// POUs/FB_NVRAM_Manager
FUNCTION_BLOCK FB_NVRAM_Manager
VAR_INPUT
    VI_Command                  : BYTE; // 1=WRITE, 2=READ, 3=FORMAT
    VI_RecordIndex              : INT;
    VI_DataPtr                  : POINTER TO BYTE;
    VI_DataSize                 : UDINT; // КРИТИЧНО: используем этот размер вместо SIZEOF
    VI_System_Time_MS           : UDINT;
    VI_Operator_ID              : STRING(10);
    VI_IsActivePLC              : BOOL;
    VI_TwoPersonConfirmation    : BOOL;
END_VAR
VAR_OUTPUT
    VO_Done                     : BOOL;
    VO_Error                    : UDINT;
    VO_ErrorID                  : UDINT;
    VO_ReadDataPtr              : POINTER TO BYTE;
    VO_HMI_Status_Message       : STRING(200);
END_VAR
VAR
    L_state                     : BYTE;
    L_step                      : UDINT;
    L_temp_buffer               : ARRAY[1..132] OF BYTE;
    L_crc32                     : FB_CRC32_Calculator;
    L_confirm_start_time        : UDINT;
    L_cmd_copy                  : BYTE;
    L_prev_Command              : BYTE;
    L_i                         : UDINT;
    L_current_time              : UDINT;
    L_cmd_rising                : BOOL;
    L_data_crc                  : DWORD;
    L_FileHandle                : RTS_IEC_HANDLE;
    L_FileName                  : STRING := '/home/root/nvram_data.bin';
    L_FileResult                : RTS_IEC_RESULT;
    L_BytesProcessed            : UDINT;
    L_BackupIdx                 : INT := 1; // Для ротации
    L_Offset                    : DINT;
END_VAR
VAR CONSTANT
    C_MAGIC_NUMBER              : UDINT := 16#534D5254; // "SMRT"
    C_STRUCT_VERSION            : UINT := 21; // ТЗ v21.0
    C_NVRAM_BASE_ADDR           : UDINT := 16#20000;
    C_HEADER_SIZE               : UDINT := 12;
    C_RECORD_SIZE               : UDINT := 128;
    C_RECORD_TOTAL_SIZE         : UDINT := 132;
    C_MAX_RECORDS               : UDINT := 96;
    C_TWO_PERSON_TIMEOUT_MS     : UDINT := 120000;
END_VAR

// Логика выполнения
L_current_time := VI_System_Time_MS;

// Детекция фронта команды
L_cmd_rising := (VI_Command <> 0) AND (L_prev_Command = 0);
L_prev_Command := VI_Command;

CASE L_state OF
    0: // ОЖИДАНИЕ (IDLE)
        IF L_cmd_rising THEN
            VO_Done := FALSE;
            VO_Error := 0;
            
            // Валидация индекса
            IF (VI_RecordIndex < 1) OR (TO_UDINT(VI_RecordIndex) > C_MAX_RECORDS) THEN
                VO_Error := 16#1501;
                VO_HMI_Status_Message := 'NVRAM: Неверный индекс записи';
                VO_Done := TRUE;
                RETURN;
            END_IF;

            // Валидация указателя
            IF VI_DataPtr = 0 THEN
                VO_Error := 16#150A;
                VO_HMI_Status_Message := 'NVRAM: Нулевой указатель данных';
                VO_Done := TRUE;
                RETURN;
            END_IF;

            IF VI_Command = 1 THEN // ЗАПИСЬ (WRITE)
                IF NOT VI_IsActivePLC THEN
                    VO_Error := 16#1509;
                    VO_HMI_Status_Message := 'NVRAM: Запись запрещена (STANDBY)';
                    VO_Done := TRUE;
                ELSIF VI_DataSize > C_RECORD_SIZE THEN
                    VO_Error := 16#150B;
                    VO_HMI_Status_Message := 'NVRAM: Размер данных больше 128 байт';
                    VO_Done := TRUE;
                ELSE
                    L_state := 1; // Переход к записи
                    L_step := 0;
                END_IF;
            ELSIF VI_Command = 2 THEN // ЧТЕНИЕ (READ)
                L_state := 2; // Переход к чтению
                L_step := 0;
            END_IF;
        END_IF;

    1: // ЗАПИСЬ_ЗАПИСИ (WRITE_RECORD)
        CASE L_step OF
            0: // Подготовка буфера и расчет CRC
                FOR L_i := 0 TO C_RECORD_SIZE - 1 DO
                    IF L_i < VI_DataSize THEN
                        L_temp_buffer[TO_INT(L_i + 1)] := VI_DataPtr[TO_INT(L_i)];
                    ELSE
                        L_temp_buffer[TO_INT(L_i + 1)] := 16#00;
                    END_IF;
                END_FOR;
                L_data_crc := L_crc32.Calculate(ADR(L_temp_buffer[1]), C_RECORD_SIZE);
                L_step := 1;
                
            1: // Открытие файла для записи
                L_FileHandle := SysFileOpen(L_FileName, AM_WRITE, ADR(L_FileResult));
                IF L_FileResult = 0 THEN
                    L_step := 2;
                ELSE
                    VO_Error := 16#150C;
                    L_state := 0;
                END_IF;
                
            2: // Позиционирование и запись
                L_Offset := TO_DINT(VI_RecordIndex - 1) * TO_DINT(C_RECORD_TOTAL_SIZE);
                L_FileResult := SysFileSetPos(L_FileHandle, TO_UDINT(L_Offset));
                L_BytesProcessed := TO_UDINT(SysFileWrite(L_FileHandle, ADR(L_temp_buffer[1]), TO_UDINT(C_RECORD_TOTAL_SIZE), ADR(L_FileResult)));
                L_FileResult := SysFileClose(L_FileHandle);
                VO_Done := TRUE;
                L_state := 0;
        END_CASE;

    2: // ЧТЕНИЕ_ЗАПИСИ (READ_RECORD)
        CASE L_step OF
            0: // Открытие файла для чтения
                L_FileHandle := SysFileOpen(L_FileName, AM_READ, ADR(L_FileResult));
                IF L_FileResult = 0 THEN
                    L_step := 1;
                ELSE
                    VO_Error := 16#150D;
                    L_state := 0;
                END_IF;
                
            1: // Чтение данных
                L_Offset := TO_DINT(VI_RecordIndex - 1) * TO_DINT(C_RECORD_TOTAL_SIZE);
                L_FileResult := SysFileSetPos(L_FileHandle, TO_UDINT(L_Offset));
                L_BytesProcessed := TO_UDINT(SysFileRead(L_FileHandle, ADR(L_temp_buffer[1]), TO_UDINT(C_RECORD_TOTAL_SIZE), ADR(L_FileResult)));
                L_FileResult := SysFileClose(L_FileHandle);
                
                // Копирование в выходной указатель
                FOR L_i := 0 TO C_RECORD_SIZE - 1 DO
                    IF L_i < VI_DataSize THEN
                        VI_DataPtr[TO_INT(L_i)] := L_temp_buffer[TO_INT(L_i + 1)];
                    END_IF;
                END_FOR;
                VO_ReadDataPtr := VI_DataPtr;
                VO_Done := TRUE;
                L_state := 0;
        END_CASE;
END_CASE;

END_FUNCTION_BLOCK

// POUs/FB_CRC32_Calculator
FUNCTION_BLOCK FB_CRC32_Calculator
VAR
    L_Table : ARRAY[0..255] OF DWORD;
    L_Initialized : BOOL := FALSE;
    L_i : INT;
    L_j : INT;
    L_Entry : DWORD;
END_VAR

METHOD Calculate : DWORD
VAR_INPUT
    VI_DataPtr : POINTER TO BYTE;
    VI_Size : UDINT;
END_VAR
VAR
    L_k : UDINT;
    L_CRC : DWORD := 16#FFFFFFFF;
END_VAR
InitTable();

IF VI_DataPtr = 0 OR VI_Size = 0 THEN
    Calculate := 0;
    RETURN;
END_IF;

FOR L_k := 0 TO VI_Size - 1 DO
    L_CRC := L_Table[TO_INT((L_CRC XOR VI_DataPtr[TO_INT(L_k)]) AND 16#FF)] XOR SHR(L_CRC, 8);
END_FOR;

Calculate := L_CRC XOR 16#FFFFFFFF;
END_METHOD

METHOD PRIVATE InitTable
VAR_INPUT
END_VAR
IF L_Initialized THEN RETURN; END_IF;

FOR L_i := 0 TO 255 DO
    L_Entry := TO_DWORD(L_i);
    FOR L_j := 0 TO 7 DO
        IF (L_Entry AND 1) <> 0 THEN
            L_Entry := SHR(L_Entry, 1) XOR 16#EDB88320;
        ELSE
            L_Entry := SHR(L_Entry, 1);
        END_IF;
    END_FOR;
    L_Table[L_i] := L_Entry;
END_FOR;
L_Initialized := TRUE;
END_METHOD

END_FUNCTION_BLOCK

// POUs/FB_Gateway_Interface
FUNCTION_BLOCK FB_Gateway_Interface
VAR_INPUT
    VI_System_Time_MS           : UDINT;
    VI_Local_PLC_Role           : E_PLC_ROLE;
    VI_Incoming_Command         : ST_Gateway_Command;
    VI_Command_Received         : BOOL;
    
    // Состояния системы
    VI_FloorHeating_Temps       : ARRAY[1..16] OF REAL;
    VI_Room_Temps               : ARRAY[1..16] OF REAL;
    VI_Zone_Valve_States        : ARRAY[1..16] OF BOOL;
    VI_Manifold_Pressures       : ARRAY[1..5] OF REAL;
    VI_Manifold_Pump_States     : ARRAY[1..5] OF BOOL;
    VI_Outdoor_Temp             : REAL;
    VI_Security_Armed           : BOOL;
    VI_Flood_Alarm_Active       : BOOL;
    VI_Gas_Alarm_Active         : BOOL;
    VI_Fire_Alarm_Active        : BOOL;
    VI_Methane_Concentration    : REAL;
    VI_Lighting_Base_Levels     : ARRAY[1..16] OF BYTE;
    VI_Socket_States            : ARRAY[1..36] OF BOOL;
    VI_Blinds_Positions         : ARRAY[1..20] OF BYTE;
    VI_Active_Scenario          : E_SCENARIO_TYPE;
END_VAR

VAR_OUTPUT
    VO_Modbus_Registers         : ARRAY[0..200] OF WORD; // Расширенный диапазон
    VO_Lighting_Override        : ARRAY[1..16] OF BYTE;
    VO_Socket_Override          : ARRAY[1..36] OF BOOL;
    VO_Data_Ready               : BOOL;
    VO_HMI_Status_Message       : STRING(200);
END_VAR

VAR
    L_last_update_time          : UDINT;
    L_i                         : INT;
    L_j                         : INT;
    L_idx                       : INT;
    L_tmp_word                  : WORD;
END_VAR

// Обновление данных Modbus (раз в 1 сек)
IF (VI_System_Time_MS - L_last_update_time) >= 1000 THEN
    L_last_update_time := VI_System_Time_MS;
    
    // 0: Статус ПЛК и Аварии
    L_tmp_word := 0;
    IF VI_Local_PLC_Role = E_PLC_ROLE.ROLE_ACTIVE THEN L_tmp_word := L_tmp_word OR 1; END_IF;
    IF VI_Security_Armed THEN L_tmp_word := L_tmp_word OR 2; END_IF;
    IF VI_Flood_Alarm_Active THEN L_tmp_word := L_tmp_word OR 4; END_IF;
    IF VI_Gas_Alarm_Active THEN L_tmp_word := L_tmp_word OR 8; END_IF;
    IF VI_Fire_Alarm_Active THEN L_tmp_word := L_tmp_word OR 16; END_IF;
    VO_Modbus_Registers[0] := L_tmp_word;

    // 1-16: Температуры пола (x10)
    FOR L_i := 1 TO 16 DO
        VO_Modbus_Registers[L_i] := TO_WORD(TO_INT(VI_FloorHeating_Temps[L_i] * 10.0));
    END_FOR;

    // 17-32: Температуры помещений (x10)
    FOR L_i := 1 TO 16 DO
        VO_Modbus_Registers[16 + L_i] := TO_WORD(TO_INT(VI_Room_Temps[L_i] * 10.0));
    END_FOR;

    // 33: Состояние клапанов зон (битовая маска 1-16)
    L_tmp_word := 0;
    FOR L_i := 1 TO 16 DO
        IF VI_Zone_Valve_States[L_i] THEN
            L_tmp_word := L_tmp_word OR SHL(TO_WORD(1), L_i - 1);
        END_IF;
    END_FOR;
    VO_Modbus_Registers[33] := L_tmp_word;

    // 34-38: Давление в коллекторах (x100)
    FOR L_i := 1 TO 5 DO
        VO_Modbus_Registers[33 + L_i] := TO_WORD(TO_INT(VI_Manifold_Pressures[L_i] * 100.0));
    END_FOR;

    // 40-55: Базовое освещение
    FOR L_i := 1 TO 16 DO
        VO_Modbus_Registers[39 + L_i] := TO_WORD(VI_Lighting_Base_Levels[L_i]);
    END_FOR;

    // 60-79: Положение штор (20 шт)
    FOR L_i := 1 TO 20 DO
        VO_Modbus_Registers[59 + L_i] := TO_WORD(VI_Blinds_Positions[L_i]);
    END_FOR;

    // 80-82: Розетки (битовая маска, 36 розеток -> 3 WORD)
    FOR L_i := 0 TO 2 DO
        L_tmp_word := 0;
        FOR L_j := 1 TO 16 DO
            L_idx := (L_i * 16) + L_j;
            IF L_idx <= 36 THEN
                IF VI_Socket_States[L_idx] THEN
                    L_tmp_word := L_tmp_word OR SHL(TO_WORD(1), L_j - 1);
                END_IF;
            END_IF;
        END_FOR;
        VO_Modbus_Registers[79 + L_i] := L_tmp_word;
    END_FOR;

    VO_Data_Ready := TRUE;
END_IF;

// Обработка входящих команд
IF VI_Command_Received AND (VI_Local_PLC_Role = E_PLC_ROLE.ROLE_ACTIVE) THEN
    CASE VI_Incoming_Command.command_type OF
        1: // Управление сценариями
            GVL_Vars.G_Current_Scenario := VI_Incoming_Command.target_scenario;
            VO_HMI_Status_Message := 'Gateway: Сценарий изменен';
        2: // Управление освещением
            IF (VI_Incoming_Command.target_zone >= 1) AND (VI_Incoming_Command.target_zone <= 16) THEN
                VO_Lighting_Override[VI_Incoming_Command.target_zone] := TO_BYTE(VI_Incoming_Command.target_value);
                VO_HMI_Status_Message := 'Gateway: Команда освещения принята';
            END_IF;
        3: // Розетки
            IF (VI_Incoming_Command.target_zone >= 1) AND (VI_Incoming_Command.target_zone <= 36) THEN
                VO_Socket_Override[VI_Incoming_Command.target_zone] := VI_Incoming_Command.target_on_off;
            END_IF;
        4: // Охрана
            // Логика постановки/снятия через PIN в FB_Security_System_Manager
            // Здесь можно только передать запрос
            VO_HMI_Status_Message := 'Gateway: Запрос охраны принят';
    END_CASE;
END_IF;

END_FUNCTION_BLOCK

// POUs/FB_Debug_Logger
FUNCTION_BLOCK FB_Debug_Logger
VAR_INPUT
    VI_Config           : ST_Debug_Logger_Config;
    VI_System_Time_MS   : UDINT;
    VI_Floor_Temps      : ARRAY[1..16] OF REAL;
    VI_Pump_Currents    : ARRAY[1..5] OF REAL;
    VI_Error_Code       : UDINT;
END_VAR
VAR
    L_buffer            : ARRAY[1..1000] OF ST_Debug_Log_Record;
    L_write_idx         : INT := 1;
    L_last_log_time     : UDINT;
    L_i                 : INT;
END_VAR

// Цикл логирования
IF VI_Config.enabled AND (VI_System_Time_MS - L_last_log_time >= VI_Config.sampling_period_ms) THEN
    L_last_log_time := VI_System_Time_MS;
    
    // Логируем температуры (если изменились или по таймауту)
    FOR L_i := 1 TO 16 DO
        L_buffer[L_write_idx].timestamp_ms := VI_System_Time_MS;
        L_buffer[L_write_idx].level := E_Debug_Log_Level.LOG_LEVEL_VERBOSE;
        L_buffer[L_write_idx].source_id := TO_BYTE(L_i);
        L_buffer[L_write_idx].value_real := VI_Floor_Temps[L_i];
        L_buffer[L_write_idx].text := 'Floor Temp Update';
        
        L_write_idx := (L_write_idx MOD 1000) + 1;
    END_FOR;

    // Логируем ошибки
    IF VI_Error_Code <> 0 THEN
        L_buffer[L_write_idx].timestamp_ms := VI_System_Time_MS;
        L_buffer[L_write_idx].level := E_Debug_Log_Level.LOG_LEVEL_MINIMAL;
        L_buffer[L_write_idx].event_code := TO_WORD(VI_Error_Code);
        L_buffer[L_write_idx].text := 'System Error Detected';
        L_write_idx := (L_write_idx MOD 1000) + 1;
    END_IF;
END_IF;

END_FUNCTION_BLOCK

// PLC_A/Application/PRG_PLC_B
PROGRAM PRG_PLC_B
VAR
    L_PLC_ID : BYTE := 2;
END_VAR

// Для ПЛК B: если он активен, G_Active_PLC_ID := 2
PRG_Main();

END_PROGRAM

// IValveController
INTERFACE IValveController

METHOD CloseValve : BOOL
VAR_INPUT
    VI_Operator_ID : STRING(10);
    VI_Force : BOOL;
END_VAR
END_METHOD

METHOD GetStatus : BYTE
VAR_INPUT
END_VAR
END_METHOD

METHOD OpenValve : BOOL
VAR_INPUT
    VI_Operator_ID : STRING(10);
    VI_Force : BOOL;
END_VAR
END_METHOD

END_INTERFACE

// POUs/FB_AccessCode_Manager
FUNCTION_BLOCK FB_AccessCode_Manager
VAR_INPUT
    VI_System_Time_MS : UDINT;
    VI_IsActivePLC    : BOOL;
    VI_Code_To_Check  : STRING(4);
END_VAR
VAR_OUTPUT
    VO_Code_Valid     : BOOL;
END_VAR
VAR
    L_Codes : ARRAY[1..5] OF STRING(4) := ['1234', '5678', '0000', '1111', '2222'];
    L_i : INT;
END_VAR

VO_Code_Valid := FALSE;
FOR L_i := 1 TO 5 DO
    IF L_Codes[L_i] = VI_Code_To_Check THEN
        VO_Code_Valid := TRUE;
        RETURN;
    END_IF;
END_FOR;

END_FUNCTION_BLOCK

// POUs/FB_Astro_Timer
FUNCTION_BLOCK FB_Astro_Timer
VAR_INPUT
    VI_System_Time_MS : UDINT;
    VI_Latitude : REAL := 55.75; // Москва
    VI_Longitude : REAL := 37.61;
END_VAR
VAR_OUTPUT
    VO_Sunset_Time : TOD;
    VO_Sunrise_Time : TOD;
    VO_Is_Night : BOOL;
END_VAR
VAR
    L_Current_TOD : TOD;
END_VAR

// Упрощенная логика астро-таймера (ТЗ 15.2)
// В реальном проекте используется библиотека SysTimeRtc или расчет по формулам
L_Current_TOD := UDINT_TO_TOD(VI_System_Time_MS MOD 86400000);

// Примерные значения для средней полосы
VO_Sunrise_Time := TOD#06:00;
VO_Sunset_Time := TOD#18:00;

// ТЗ 15.2: Закат + 30 мин / Рассвет - 30 мин
VO_Is_Night := (L_Current_TOD > (VO_Sunset_Time + T#30m)) OR (L_Current_TOD < (VO_Sunrise_Time - T#30m));

END_FUNCTION_BLOCK

// POUs/FB_BlackBox_Recorder
FUNCTION_BLOCK FB_BlackBox_Recorder
VAR_INPUT
    VI_Current_Data : ST_BlackBox_Record;
    VI_Freeze       : BOOL;
END_VAR
VAR
    L_Write_Index   : INT := 0;
    L_FileHandle    : RTS_IEC_HANDLE;
    L_FileName      : STRING := '/home/root/blackbox_dump.bin';
    L_FileResult    : RTS_IEC_RESULT;
    L_State         : INT;
END_VAR

CASE L_State OF
    0: // Циклическая запись
        IF NOT G_BlackBox_Frozen THEN
            G_BlackBox_Buffer[L_Write_Index] := VI_Current_Data;
            G_BlackBox_LastIndex := L_Write_Index;
            
            L_Write_Index := L_Write_Index + 1;
            IF L_Write_Index > 99 THEN
                L_Write_Index := 0;
            END_IF;
            
            IF VI_Freeze THEN
                G_BlackBox_Frozen := TRUE;
                L_State := 1;
            END_IF;
        END_IF;
        
    1: // Сохранение на Flash (SD-карту или внутреннюю память ПЛК210)
        L_FileHandle := SysFileOpen(L_FileName, AM_WRITE, ADR(L_FileResult));
        IF L_FileResult = 0 THEN
            SysFileWrite(L_FileHandle, ADR(G_BlackBox_Buffer[0]), SIZEOF(G_BlackBox_Buffer), ADR(L_FileResult));
            SysFileClose(L_FileHandle);
            L_State := 2;
        END_IF;
        
    2: // Завершено
        ;
END_CASE;

END_FUNCTION_BLOCK

// POUs/FB_Boiler_Cascade_Controller
FUNCTION_BLOCK FB_Boiler_Cascade_Controller
VAR_INPUT
    VI_Demand_kW : REAL;
    VI_IsActivePLC : BOOL;
END_VAR
VAR_OUTPUT
    VO_Boiler1_On : BOOL;
    VO_Boiler2_On : BOOL;
END_VAR
VAR
    L_Lead_Boiler : BYTE := 1; // 1 или 2
    L_Boiler1_Hours : UDINT;
    L_Boiler2_Hours : UDINT;
    L_Last_Hour_Update : UDINT;
    L_System_Time : UDINT;
END_VAR
VAR_INPUT
    VI_System_Time : UDINT;
END_VAR

// Логика ротации по наработке
IF (VI_System_Time - L_Last_Hour_Update) >= 3600000 THEN // Раз в час
    L_Last_Hour_Update := VI_System_Time;
    IF VO_Boiler1_On THEN L_Boiler1_Hours := L_Boiler1_Hours + 1; END_IF;
    IF VO_Boiler2_On THEN L_Boiler2_Hours := L_Boiler2_Hours + 1; END_IF;
    
    // Смена ведущего, если разница более 100 часов
    IF (L_Boiler1_Hours > L_Boiler2_Hours + 100) THEN
        L_Lead_Boiler := 2;
    ELSIF (L_Boiler2_Hours > L_Boiler1_Hours + 100) THEN
        L_Lead_Boiler := 1;
    END_IF;
END_IF;

IF VI_IsActivePLC THEN
    IF VI_Demand_kW > 24.0 THEN
        VO_Boiler1_On := TRUE;
        VO_Boiler2_On := TRUE;
    ELSIF VI_Demand_kW > 2.0 THEN
        VO_Boiler1_On := (L_Lead_Boiler = 1);
        VO_Boiler2_On := (L_Lead_Boiler = 2);
    ELSE
        VO_Boiler1_On := FALSE;
        VO_Boiler2_On := FALSE;
    END_IF;
END_IF;

END_FUNCTION_BLOCK

// POUs/FB_Boiler_Cascade_Manager
FUNCTION_BLOCK FB_Boiler_Cascade_Manager
VAR_INPUT
    VI_Boiler1_Status : ST_Boiler_Status;
    VI_Boiler2_Status : ST_Boiler_Status;
    VI_Role_Swap_Interval : UDINT := 168; // часы
END_VAR
VAR_OUTPUT
    VO_Boiler1_Enable : BOOL;
    VO_Boiler2_Enable : BOOL;
END_VAR

// Логика п. 2.8: Включение резервного при >80% мощности или отказе
IF VI_Boiler1_Status.Error OR VI_Boiler1_Status.Current_Power > 80.0 THEN
    VO_Boiler2_Enable := TRUE;
ELSE
    VO_Boiler2_Enable := FALSE;
END_IF;

VO_Boiler1_Enable := NOT VI_Boiler1_Status.Error;

END_FUNCTION_BLOCK

// POUs/FB_Calibration_Manager
FUNCTION_BLOCK FB_Calibration_Manager
VAR_INPUT
    VI_Raw_Value : REAL;
    VI_Type : BYTE; // 1-Temp, 2-Pressure, 3-Gas
    VI_Calib_Record : ST_Sensor_Calibration_Record;
    VI_System_Time_MS : UDINT;
    VI_Start_Verification : BOOL;
END_VAR
VAR_OUTPUT
    VO_Calibrated_Value : REAL;
    VO_Verification_Active : BOOL;
    VO_Verification_Failed : BOOL;
    VO_Deviation_Percent : REAL;
END_VAR
VAR
    L_Verification_Timer : TON;
    L_Initial_Value : REAL;
END_VAR

// 1. Расчет калиброванного значения
CASE VI_Type OF
    1: VO_Calibrated_Value := VI_Raw_Value + VI_Calib_Record.offset;
    2, 3: VO_Calibrated_Value := (VI_Raw_Value * VI_Calib_Record.multiplier) + VI_Calib_Record.offset;
END_CASE;

// 2. Верификация через 1 час (ТЗ 9.5)
IF VI_Start_Verification AND NOT VO_Verification_Active THEN
    VO_Verification_Active := TRUE;
    L_Initial_Value := VO_Calibrated_Value;
    L_Verification_Timer(IN := TRUE, PT := T#1h);
END_IF;

L_Verification_Timer(IN := VO_Verification_Active);

IF L_Verification_Timer.Q THEN
    VO_Verification_Active := FALSE;
    L_Verification_Timer(IN := FALSE);
    
    // ТЗ 9.5: Отклонение ≤2.0% (норма) / >5.0% (ошибка)
    IF L_Initial_Value <> 0 THEN
        VO_Deviation_Percent := ABS(VO_Calibrated_Value - L_Initial_Value) / L_Initial_Value * 100.0;
    ELSE
        VO_Deviation_Percent := 0.0;
    END_IF;
    
    VO_Verification_Failed := (VO_Deviation_Percent > 5.0);
END_IF;

END_FUNCTION_BLOCK

// POUs/FB_CO_Detector
FUNCTION_BLOCK FB_CO_Detector
VAR_INPUT
    VI_CO_PPM : REAL;
    VI_Threshold_Warning : REAL := 30.0;
    VI_Threshold_Alarm   : REAL := 70.0;
END_VAR
VAR_OUTPUT
    VO_Warning_Active : BOOL;
    VO_Alarm_Active   : BOOL;
END_VAR

VO_Warning_Active := (VI_CO_PPM >= VI_Threshold_Warning);
VO_Alarm_Active := (VI_CO_PPM >= VI_Threshold_Alarm);

END_FUNCTION_BLOCK

// POUs/FB_Device_Predictive_Diag
FUNCTION_BLOCK FB_Device_Predictive_Diag
VAR_INPUT
    VI_Current_Value : REAL;      // Текущий ток или время
    VI_Nominal_Value : REAL;      // Эталонное значение
    VI_Is_Running    : BOOL;
    VI_Reset_Stats   : BOOL;
END_VAR
VAR_IN_OUT
    VIO_Health_Data  : ST_Device_Health;
END_VAR
VAR
    L_Prev_Running   : BOOL;
    L_Current_Sum    : REAL;
    L_Sample_Count   : UDINT;
END_VAR

// 1. Счётчик пусков и замер пускового тока
IF VI_Is_Running AND NOT L_Prev_Running THEN
    VIO_Health_Data.Starts_Count := VIO_Health_Data.Starts_Count + 1;
    VIO_Health_Data.Last_Start_Current := VI_Current_Value;
    
    // Обновление среднего пускового тока
    L_Sample_Count := L_Sample_Count + 1;
    L_Current_Sum := L_Current_Sum + VI_Current_Value;
    VIO_Health_Data.Avg_Start_Current := L_Current_Sum / UDINT_TO_REAL(L_Sample_Count);
END_IF;

// 2. Анализ отклонения (п. 12.1 ТЗ)
IF VI_Is_Running THEN
    // Если ток выше номинала на 50% - снижаем здоровье
    IF VI_Current_Value > (VI_Nominal_Value * 1.5) THEN
        IF VIO_Health_Data.Health_Score > 0 THEN
            VIO_Health_Data.Health_Score := VIO_Health_Data.Health_Score - 1;
        END_IF;
    END_IF;
END_IF;

// 3. Генерация предупреждения
IF VIO_Health_Data.Health_Score < 20 THEN
    VIO_Health_Data.Maintenance_Required := TRUE;
    VIO_Health_Data.Warning_Message := 'Критический износ: проверьте механику';
ELSIF VIO_Health_Data.Health_Score < 60 THEN
    VIO_Health_Data.Warning_Message := 'Предупреждение: повышенное трение';
END_IF;

L_Prev_Running := VI_Is_Running;

END_FUNCTION_BLOCK

// POUs/FB_Emergency_Valve_Open
FUNCTION_BLOCK FB_Emergency_Valve_Open
VAR_INPUT
    VI_Fire_Alarm : BOOL;
    VI_Gas_Alarm  : BOOL;
END_VAR
VAR_OUTPUT
    VO_Open_Cmd   : BOOL;
END_VAR

// Приоритетное открытие при любой серьезной аварии
VO_Open_Cmd := VI_Fire_Alarm OR VI_Gas_Alarm;

END_FUNCTION_BLOCK

// POUs/FB_Exhaust_Ventilation_Controller
FUNCTION_BLOCK FB_Exhaust_Ventilation_Controller
VAR_INPUT
    VI_Humidity : REAL;
    VI_CO2      : REAL;
    VI_Config   : ST_Ventilation_Unit_Config;
END_VAR
VAR_OUTPUT
    VO_Fan_Speed : BYTE;
END_VAR

IF VI_Humidity > VI_Config.Threshold_Hum THEN
    VO_Fan_Speed := 100;
ELSIF VI_CO2 > 800.0 THEN
    VO_Fan_Speed := 70;
ELSE
    VO_Fan_Speed := 40;
END_IF;

END_FUNCTION_BLOCK

// POUs/FB_Flood_Detector
FUNCTION_BLOCK FB_Flood_Detector
VAR_INPUT
    VI_Sensors : ARRAY[1..12] OF BOOL;
    VI_IsActivePLC : BOOL;
END_VAR
VAR_OUTPUT
    VO_Flood_Alarm : BOOL;
    VO_Close_Valve_35 : BOOL;
    VO_Close_Valve_36 : BOOL;
END_VAR
VAR
    L_i : INT;
END_VAR

VO_Flood_Alarm := FALSE;
VO_Close_Valve_35 := FALSE;
VO_Close_Valve_36 := FALSE;

FOR L_i := 1 TO 12 DO
    IF VI_Sensors[L_i] THEN
        VO_Flood_Alarm := TRUE;
        IF VI_IsActivePLC THEN
            // Логика п. 4.2: Зона 2 (4-5) и Зона 3 (6-7) делят клапан 36
            IF L_i >= 4 AND L_i <= 7 THEN
                VO_Close_Valve_36 := TRUE;
            ELSIF L_i >= 1 AND L_i <= 3 THEN
                VO_Close_Valve_35 := TRUE;
            END_IF;
        END_IF;
    END_IF;
END_FOR;

END_FUNCTION_BLOCK

// POUs/FB_FloorHeating_Controller
FUNCTION_BLOCK FB_FloorHeating_Controller
VAR_INPUT
    VI_Current_Temp : REAL;
    VI_Config : ST_FloorHeating_Circuit_Config;
    VI_Tariff : ST_Tariff_Config;
    VI_Current_Hour : UINT;
    VI_IsActivePLC : BOOL;
END_VAR
VAR_OUTPUT
    VO_Pump_Run : BOOL;
    VO_Valve_Pos : REAL; // 0..10V
    VO_Effective_Setpoint : REAL;
END_VAR
VAR
    L_Is_Night : BOOL;
END_VAR

// 1. Определение активного тарифа
IF VI_Tariff.Enabled THEN
    IF VI_Tariff.Night_Start_Hour > VI_Tariff.Night_End_Hour THEN
        // Переход через полночь (например, 23:00 - 07:00)
        L_Is_Night := (VI_Current_Hour >= VI_Tariff.Night_Start_Hour) OR (VI_Current_Hour < VI_Tariff.Night_End_Hour);
    ELSE
        // В пределах одного дня
        L_Is_Night := (VI_Current_Hour >= VI_Tariff.Night_Start_Hour) AND (VI_Current_Hour < VI_Tariff.Night_End_Hour);
    END_IF;
ELSE
    L_Is_Night := FALSE;
END_IF;

// 2. Расчет эффективной уставки
VO_Effective_Setpoint := VI_Config.design_temp;
IF L_Is_Night THEN
    VO_Effective_Setpoint := VO_Effective_Setpoint + VI_Tariff.Boost_Delta;
END_IF;

// 3. Простая логика управления (гистерезис)
IF VI_IsActivePLC THEN
    IF VI_Current_Temp < (VO_Effective_Setpoint - 0.5) THEN
        VO_Pump_Run := TRUE;
        VO_Valve_Pos := 10.0;
    ELSIF VI_Current_Temp > (VO_Effective_Setpoint + 0.5) THEN
        VO_Pump_Run := FALSE;
        VO_Valve_Pos := 0.0;
    END_IF;
END_IF;

END_FUNCTION_BLOCK

// POUs/FB_FloorHeating_Freeze_Protection
FUNCTION_BLOCK FB_FloorHeating_Freeze_Protection
VAR_INPUT
    VI_Floor_Temps : ARRAY[1..16] OF REAL;
    VI_Outdoor_Temp : REAL;
    VI_Threshold : REAL := 7.0;
END_VAR
VAR_OUTPUT
    VO_Freeze_Alert : BOOL;
    VO_Pump_Force_On : BOOL;
END_VAR
VAR
    L_i : INT;
END_VAR

VO_Freeze_Alert := FALSE;
VO_Pump_Force_On := FALSE;

FOR L_i := 1 TO 16 DO
    IF VI_Floor_Temps[L_i] < VI_Threshold THEN
        VO_Freeze_Alert := TRUE;
        VO_Pump_Force_On := TRUE;
        RETURN;
    END_IF;
END_FOR;

IF VI_Outdoor_Temp < -5.0 THEN
    VO_Pump_Force_On := TRUE;
END_IF;

END_FUNCTION_BLOCK

// POUs/FB_FloorHeating_Overheat_Protection
FUNCTION_BLOCK FB_FloorHeating_Overheat_Protection
VAR_INPUT
    VI_Temps : ARRAY[1..16] OF REAL;
    VI_Threshold : REAL := 45.0;
END_VAR
VAR_OUTPUT
    VO_Overheat_Detected : BOOL;
    VO_Locked_Circuits : ARRAY[1..16] OF BOOL;
END_VAR
VAR
    L_i : INT;
END_VAR

VO_Overheat_Detected := FALSE;
FOR L_i := 1 TO 16 DO
    IF VI_Temps[L_i] > VI_Threshold THEN
        VO_Overheat_Detected := TRUE;
        VO_Locked_Circuits[L_i] := TRUE;
    END_IF;
END_FOR;

END_FUNCTION_BLOCK

// POUs/FB_Gas_Methane_Detector
FUNCTION_BLOCK FB_Gas_Methane_Detector
VAR_INPUT
    VI_Methane_LEL : REAL;
    VI_Threshold_Alarm : REAL := 20.0;
END_VAR
VAR_OUTPUT
    VO_Alarm_Active : BOOL;
    VO_Close_Valve  : BOOL;
END_VAR

VO_Alarm_Active := (VI_Methane_LEL >= VI_Threshold_Alarm);
VO_Close_Valve := VO_Alarm_Active;

END_FUNCTION_BLOCK

// POUs/FB_Gas_Valve_Controller
FUNCTION_BLOCK FB_Gas_Valve_Controller IMPLEMENTS IValveController
VAR_INPUT
    VI_System_Time : UDINT;
    VI_IsActivePLC : BOOL;
    VI_Gas_Alarm   : BOOL;
    VI_Config      : ST_Gas_Valve_Configuration;
END_VAR
VAR_OUTPUT
    VO_Valve_Closed : BOOL;
    VO_Status_Msg   : STRING(200);
END_VAR

// При аварии газа - немедленное закрытие
IF VI_Gas_Alarm AND VI_IsActivePLC THEN
    VO_Valve_Closed := TRUE;
    VO_Status_Msg := 'ГАЗОВЫЙ КЛАПАН ЗАКРЫТ ПО АВАРИИ';
END_IF;

METHOD CloseValve : BOOL
VAR_INPUT
    VI_Operator_ID : STRING(10);
    VI_Force : BOOL;
END_VAR
VO_Valve_Closed := TRUE;
CloseValve := TRUE;
END_METHOD

METHOD GetStatus : BYTE
VAR_INPUT
END_VAR
GetStatus := TO_BYTE(SEL(VO_Valve_Closed, 0, 1));
END_METHOD

METHOD OpenValve : BOOL
VAR_INPUT
    VI_Operator_ID : STRING(10);
    VI_Force : BOOL;
END_VAR
IF VI_IsActivePLC OR VI_Force THEN
    VO_Valve_Closed := FALSE;
    OpenValve := TRUE;
END_IF;
END_METHOD

END_FUNCTION_BLOCK

// POUs/FB_History_Manager
FUNCTION_BLOCK FB_History_Manager
VAR_INPUT
    VI_System_Time_MS : UDINT;
    VI_Write_Event    : BOOL;
    VI_Event          : ST_History_Record;
END_VAR
VAR_OUTPUT
    VO_Total_Events   : UDINT;
END_VAR
VAR
    L_History_Buffer : ARRAY[1..100] OF ST_History_Record;
    L_Write_Idx      : INT := 1;
END_VAR

IF VI_Write_Event THEN
    L_History_Buffer[L_Write_Idx] := VI_Event;
    L_History_Buffer[L_Write_Idx].timestamp_ms := VI_System_Time_MS;
    
    L_Write_Idx := (L_Write_Idx MOD 100) + 1;
    VO_Total_Events := VO_Total_Events + 1;
END_IF;

END_FUNCTION_BLOCK

// POUs/FB_Lifetime_Predictor
FUNCTION_BLOCK FB_Lifetime_Predictor
VAR_INPUT
    VI_Runtime_Hours : UDINT;
    VI_Start_Count   : UDINT;
    VI_Nominal_Life  : UDINT := 10000;
END_VAR
VAR_OUTPUT
    VO_Remaining_Percent : BYTE;
    VO_Maintenance_Req   : BOOL;
END_VAR

// Упрощенная модель износа
IF VI_Nominal_Life > 0 THEN
    VO_Remaining_Percent := TO_BYTE(100 - (VI_Runtime_Hours * 100 / VI_Nominal_Life));
ELSE
    VO_Remaining_Percent := 0;
END_IF;

VO_Maintenance_Req := (VO_Remaining_Percent < 10);

END_FUNCTION_BLOCK

// POUs/FB_Maintenance_Access
FUNCTION_BLOCK FB_Maintenance_Access
VAR_INPUT
    VI_System_Time : UDINT;
    VI_Activate    : BOOL;
    VI_Duration    : UDINT := 60; // мин
END_VAR
VAR_OUTPUT
    VO_Active      : BOOL;
    VO_Time_Left   : UDINT;
END_VAR
VAR
    L_Start_Time   : UDINT;
    L_elapsed      : UDINT;
END_VAR

IF VI_Activate AND NOT VO_Active THEN
    VO_Active := TRUE;
    L_Start_Time := VI_System_Time;
END_IF;

IF VO_Active THEN
    L_elapsed := (VI_System_Time - L_Start_Time) / 60000;
    IF L_elapsed >= VI_Duration THEN
        VO_Active := FALSE;
    ELSE
        VO_Time_Left := VI_Duration - L_elapsed;
    END_IF;
END_IF;

END_FUNCTION_BLOCK

// POUs/FB_Manifold_Mixing_Valve_Controller
FUNCTION_BLOCK FB_Manifold_Mixing_Valve_Controller
VAR_INPUT
    VI_Setpoint : REAL;
    VI_Actual   : REAL;
END_VAR
VAR_OUTPUT
    VO_Valve_Pos : REAL; // 0-100%
END_VAR

// ПИД-регулятор (упрощенно для примера)
VO_Valve_Pos := (VI_Setpoint - VI_Actual) * 10.0;
IF VO_Valve_Pos > 100.0 THEN VO_Valve_Pos := 100.0;
ELSIF VO_Valve_Pos < 0.0 THEN VO_Valve_Pos := 0.0;
END_IF;

END_FUNCTION_BLOCK

// POUs/FB_Manifold_Pump_Controller
FUNCTION_BLOCK FB_Manifold_Pump_Controller
VAR_INPUT
    VI_Enable_Request : BOOL;
    VI_System_Time : UDINT;
    VI_Stop_Ramp_MS : UDINT := 5000;
END_VAR
VAR_OUTPUT
    VO_Speed_Percent : BYTE;
    VO_Running : BOOL;
END_VAR
VAR
    L_Stop_Start_Time : UDINT;
    L_Stopping : BOOL;
    L_elapsed : UDINT;
END_VAR

IF VI_Enable_Request THEN
    VO_Speed_Percent := 100;
    VO_Running := TRUE;
    L_Stopping := FALSE;
ELSE
    IF VO_Running AND NOT L_Stopping THEN
        L_Stopping := TRUE;
        L_Stop_Start_Time := VI_System_Time;
    END_IF;
    
    IF L_Stopping THEN
        L_elapsed := VI_System_Time - L_Stop_Start_Time;
        IF L_elapsed < VI_Stop_Ramp_MS THEN
            // Исправлено: защита от отрицательного значения
            VO_Speed_Percent := REAL_TO_BYTE(100.0 * (1.0 - TO_REAL(L_elapsed) / TO_REAL(VI_Stop_Ramp_MS)));
        ELSE
            VO_Speed_Percent := 0;
            VO_Running := FALSE;
            L_Stopping := FALSE;
        END_IF;
    END_IF;
END_IF;

END_FUNCTION_BLOCK

// POUs/FB_Manual_Valve_Control
FUNCTION_BLOCK FB_Manual_Valve_Control
VAR_INPUT
    VI_System_Time : UDINT;
    VI_Open_Req    : BOOL;
    VI_Duration    : UDINT := 5; // мин
END_VAR
VAR_OUTPUT
    VO_Open_Cmd    : BOOL;
    VO_Time_Left   : UDINT;
END_VAR
VAR
    L_Start_Time   : UDINT;
    L_Active       : BOOL;
    L_elapsed      : UDINT;
END_VAR

// Логика ручного управления клапаном с таймером автозакрытия
IF VI_Open_Req AND NOT L_Active THEN
    L_Active := TRUE;
    L_Start_Time := VI_System_Time;
    VO_Open_Cmd := TRUE;
END_IF;

IF L_Active THEN
    // Расчет оставшегося времени в минутах
    L_elapsed := (VI_System_Time - L_Start_Time) / 60000;
    IF L_elapsed >= VI_Duration THEN
        L_Active := FALSE;
        VO_Open_Cmd := FALSE;
    ELSE
        VO_Time_Left := VI_Duration - L_elapsed;
    END_IF;
ELSE
    VO_Time_Left := 0;
END_IF;

END_FUNCTION_BLOCK

// POUs/FB_Outdoor_Lighting_Controller
FUNCTION_BLOCK FB_Outdoor_Lighting_Controller
VAR_INPUT
    VI_Ambient_Lux : REAL;
    VI_Motion      : BOOL;
    VI_Security    : BOOL;
END_VAR
VAR_OUTPUT
    VO_Light_On    : BOOL;
END_VAR

IF VI_Security AND VI_Motion THEN
    VO_Light_On := TRUE; // Тревожное освещение
ELSIF VI_Ambient_Lux < 50.0 THEN
    VO_Light_On := TRUE; // Ночное освещение
ELSE
    VO_Light_On := FALSE;
END_IF;

END_FUNCTION_BLOCK

// POUs/FB_Presence_Playback
FUNCTION_BLOCK FB_Presence_Playback
VAR_INPUT
    VI_Mode_Record : BOOL; // TRUE - записываем, FALSE - воспроизводим
    VI_Light_Inputs : ARRAY[1..16] OF BOOL;
    VI_Time_Index   : UDINT; // Индекс времени в рамках недели (мс)
END_VAR
VAR_OUTPUT
    VO_Light_Outputs : ARRAY[1..16] OF BOOL;
END_VAR
VAR
    // В ПЛК210 используем массив в памяти, который должен быть привязан к файлу на SD или NVRAM
    L_History : ARRAY[0..1007] OF WORD; // 168 часов * 6 записей в час = 1008 записей (битовая маска 16 ламп)
    L_Current_Slot : UDINT;
    L_i : INT;
END_VAR

L_Current_Slot := (VI_Time_Index / 600000) MOD 1008; // Слот каждые 10 минут

IF VI_Mode_Record THEN
    // Запись текущего состояния в слот
    L_History[L_Current_Slot] := 0;
    FOR L_i := 1 TO 16 DO
        IF VI_Light_Inputs[L_i] THEN
            L_History[L_Current_Slot] := L_History[L_Current_Slot] OR SHL(WORD#1, L_i-1);
        END_IF;
    END_FOR;
ELSE
    // Воспроизведение из слота
    FOR L_i := 1 TO 16 DO
        VO_Light_Outputs[L_i] := (L_History[L_Current_Slot] AND SHL(WORD#1, L_i-1)) <> 0;
    END_FOR;
END_IF;

END_FUNCTION_BLOCK

// POUs/FB_Presence_Simulator
FUNCTION_BLOCK FB_Presence_Simulator
VAR_INPUT
    VI_Enabled : BOOL;
    VI_Intensity : REAL; 
    VI_System_Time : UDINT;
    VI_Use_Playback : BOOL; // Новый режим воспроизведения
END_VAR
VAR_OUTPUT
    VO_Light_States : ARRAY[1..16] OF BOOL;
END_VAR
VAR
    fbPlayback : FB_Presence_Playback;
END_VAR

IF VI_Enabled THEN
    IF VI_Use_Playback THEN
        fbPlayback(VI_Mode_Record := FALSE, VI_Time_Index := VI_System_Time MOD 604800000, VO_Light_Outputs => VO_Light_States);
    ELSE
        // Старая логика случайной симуляции
        VO_Light_States[1] := (VI_System_Time MOD 100000 > 50000);
    END_IF;
END_IF;

END_FUNCTION_BLOCK

// POUs/FB_Pre_Departure_Heating
FUNCTION_BLOCK FB_Pre_Departure_Heating
VAR_INPUT
    VI_Departure_Time : UDINT;
    VI_System_Time    : UDINT;
    VI_Selected       : ARRAY[1..16] OF BOOL;
END_VAR
VAR_OUTPUT
    VO_Heating_Active : BOOL;
    VO_Setpoints      : ARRAY[1..16] OF REAL;
END_VAR

VAR
    L_i : INT;
END_VAR

// Запуск за 3 часа (10800000 мс)
IF (VI_Departure_Time - VI_System_Time) < 10800000 THEN
    VO_Heating_Active := TRUE;
    FOR L_i := 1 TO 16 DO
        IF VI_Selected[L_i] THEN VO_Setpoints[L_i] := 22.0; END_IF;
    END_FOR;
ELSE
    VO_Heating_Active := FALSE;
END_IF;

END_FUNCTION_BLOCK

// POUs/FB_Scenario_Manager
FUNCTION_BLOCK FB_Scenario_Manager
VAR_INPUT
    VI_System_Time_MS : UDINT;
    VI_Activate_Request : E_SCENARIO_TYPE;
    VI_IsActivePLC : BOOL;
END_VAR
VAR_OUTPUT
    VO_Current_Scenario : E_SCENARIO_TYPE;
    VO_Status_Msg : STRING(200);
END_VAR

IF VI_IsActivePLC AND (VI_Activate_Request <> VO_Current_Scenario) THEN
    // Логика переключения сценариев
    VO_Current_Scenario := VI_Activate_Request;
    
    CASE VO_Current_Scenario OF
        E_SCENARIO_TYPE.SCENARIO_NONE:
            VO_Status_Msg := 'Сценарии отключены';
        E_SCENARIO_TYPE.SCENARIO_AWAY:
            VO_Status_Msg := 'Активирован сценарий: Вне дома (Охрана + Энергосбережение)';
        E_SCENARIO_TYPE.SCENARIO_SLEEP:
            VO_Status_Msg := 'Активирован сценарий: Сон (Ночное освещение + Климат)';
        E_SCENARIO_TYPE.SCENARIO_PRESENCE:
            VO_Status_Msg := 'Активирован сценарий: Имитация присутствия';
    END_CASE;
END_IF;

END_FUNCTION_BLOCK

// POUs/FB_Scenario_Transition_Controller
FUNCTION_BLOCK FB_Scenario_Transition_Controller
VAR_INPUT
    VI_System_Time : UDINT;
    VI_Start_Time  : UDINT;
    VI_Min_Dur     : UDINT := 300000; // 5 мин
END_VAR
VAR_OUTPUT
    VO_Allowed     : BOOL;
END_VAR

VO_Allowed := (VI_System_Time - VI_Start_Time) >= VI_Min_Dur;

END_FUNCTION_BLOCK

// POUs/FB_Security_Alarm
FUNCTION_BLOCK FB_Security_Alarm
VAR_INPUT
    VI_IsActivePLC : BOOL;
    VI_Assigned_DoorWindow_Open : ARRAY[1..20] OF BOOL;
    VI_Assigned_GlassBreak : ARRAY[1..12] OF BOOL;
END_VAR
VAR_OUTPUT
    VO_Alarm_Active : BOOL;
    VO_Status_Msg : STRING(200);
END_VAR

VO_Alarm_Active := CheckPerimeter();

IF VO_Alarm_Active THEN
    VO_Status_Msg := 'ТРЕВОГА: НАРУШЕН ПЕРИМЕТР';
ELSE
    VO_Status_Msg := 'Периметр в норме';
END_IF;

METHOD CheckPerimeter : BOOL
VAR
    L_i : INT;
END_VAR
CheckPerimeter := FALSE;
// Проверка окон
FOR L_i := 1 TO 20 DO
    IF VI_Assigned_DoorWindow_Open[L_i] THEN
        CheckPerimeter := TRUE;
        RETURN;
    END_IF;
END_FOR;
// Проверка стекол
FOR L_i := 1 TO 12 DO
    IF VI_Assigned_GlassBreak[L_i] THEN
        CheckPerimeter := TRUE;
        RETURN;
    END_IF;
END_FOR;
END_METHOD

END_FUNCTION_BLOCK

// POUs/FB_Security_System
FUNCTION_BLOCK FB_Security_System
VAR_INPUT
    VI_System_Time : UDINT;
    VI_Sensors_Open : ARRAY[1..15] OF BOOL;
    VI_Sensors_Glass : ARRAY[1..15] OF BOOL;
    VI_Grouped_2F : BOOL;
    VI_PIN_Code : STRING(4);
    VI_Arm_Request : BOOL;
END_VAR
VAR_OUTPUT
    VO_Alarm_Active : BOOL;
    VO_Alarm_Level : E_ALERT_PRIORITY;
    VO_Status : BYTE; // 0-Disarmed, 1-Arming, 2-Armed, 3-Alarm
END_VAR
VAR
    L_Last_Trigger_Time : UDINT;
    L_Trigger_Count : INT;
    L_i : INT;
END_VAR

L_Trigger_Count := 0;
FOR L_i := 1 TO 15 DO
    IF VI_Sensors_Open[L_i] OR VI_Sensors_Glass[L_i] THEN
        L_Trigger_Count := L_Trigger_Count + 1;
    END_IF;
END_FOR;
IF VI_Grouped_2F THEN L_Trigger_Count := L_Trigger_Count + 1; END_IF;

// Логика п. 3.3: Комбинированные события (>=2 датчиков за 10 сек)
IF L_Trigger_Count >= 2 THEN
    IF (VI_System_Time - L_Last_Trigger_Time) < 10000 THEN
        VO_Alarm_Level := E_ALERT_PRIORITY.ALERT_PRIORITY_CRITICAL;
        VO_Alarm_Active := TRUE;
    END_IF;
    L_Last_Trigger_Time := VI_System_Time;
END_IF;

END_FUNCTION_BLOCK

// POUs/FB_Sensor_Calibration_Processor
FUNCTION_BLOCK FB_Sensor_Calibration_Processor
VAR_INPUT
    VI_Raw_Value : REAL;
    VI_Calib_Record : ST_Sensor_Calibration_Record;
END_VAR
VAR_OUTPUT
    VO_Calibrated_Value : REAL;
END_VAR

// Формула: (Сырое значение * Множитель) + Смещение
VO_Calibrated_Value := (VI_Raw_Value * VI_Calib_Record.multiplier) + VI_Calib_Record.offset;

END_FUNCTION_BLOCK

// POUs/FB_Sensor_Distribution
FUNCTION_BLOCK FB_Sensor_Distribution
VAR_INPUT
    VI_Local_PLC_ID : BYTE; // 1=A, 2=B
    VI_Raw_Sensors  : ARRAY[1..20] OF BOOL;
END_VAR
VAR_OUTPUT
    VO_Assigned_Sensors : ARRAY[1..20] OF BOOL;
END_VAR
VAR
    L_i : INT;
END_VAR

FOR L_i := 1 TO 20 DO
    // ПЛК A берет четные, ПЛК B - нечетные
    IF (VI_Local_PLC_ID = 1 AND (L_i MOD 2 = 0)) OR
       (VI_Local_PLC_ID = 2 AND (L_i MOD 2 <> 0)) THEN
        VO_Assigned_Sensors[L_i] := VI_Raw_Sensors[L_i];
    END_IF;
END_FOR;

END_FUNCTION_BLOCK

// POUs/FB_Smoke_Detector
FUNCTION_BLOCK FB_Smoke_Detector
VAR_INPUT
    VI_Sensors : ARRAY[1..6] OF BOOL;
    VI_System_Time : UDINT;
END_VAR
VAR_OUTPUT
    VO_Fire_Alarm : BOOL;
END_VAR
VAR
    L_Verify_Start : ARRAY[1..6] OF UDINT;
    L_Verifying    : ARRAY[1..6] OF BOOL;
    L_i : INT;
END_VAR

FOR L_i := 1 TO 6 DO
    IF VI_Sensors[L_i] THEN
        IF NOT L_Verifying[L_i] THEN
            L_Verifying[L_i] := TRUE;
            L_Verify_Start[L_i] := VI_System_Time;
        ELSIF (VI_System_Time - L_Verify_Start[L_i]) > 30000 THEN
            VO_Fire_Alarm := TRUE;
        END_IF;
    ELSE
        L_Verifying[L_i] := FALSE;
    END_IF;
END_FOR;

END_FUNCTION_BLOCK

// POUs/FB_SMS_Notification
FUNCTION_BLOCK FB_SMS_Notification
VAR_INPUT
    VI_Send_Request : BOOL;
    VI_Phone        : STRING(15);
    VI_Text         : STRING(160);
END_VAR
VAR_OUTPUT
    VO_Done         : BOOL;
    VO_Error        : BOOL;
END_VAR

VAR
    L_State : INT;
    L_Timer : TON;
    L_AT_Command : STRING(255);
END_VAR

CASE L_State OF
    0: // Ожидание запроса
        IF VI_Send_Request THEN
            VO_Done := FALSE;
            VO_Error := FALSE;
            L_State := 1;
        END_IF;
        
    1: // Отправка AT+CMGF=1 (Установка текстового режима)
        L_AT_Command := 'AT+CMGF=1$R';
        L_State := 2;
        L_Timer(IN := TRUE, PT := T#500ms);
        
    2: // Ожидание ответа OK и отправка номера
        L_Timer(IN := TRUE);
        IF L_Timer.Q THEN
            L_Timer(IN := FALSE);
            L_AT_Command := CONCAT('AT+CMGS="', CONCAT(VI_Phone, '"$R'));
            L_State := 3;
            L_Timer(IN := TRUE, PT := T#500ms);
        END_IF;
        
    3: // Отправка текста сообщения и символа Ctrl+Z (ASCII 26)
        L_Timer(IN := TRUE);
        IF L_Timer.Q THEN
            L_Timer(IN := FALSE);
            L_AT_Command := CONCAT(VI_Text, '$1A'); // $1A - это Ctrl+Z в CODESYS
            L_State := 4;
            L_Timer(IN := TRUE, PT := T#2s);
        END_IF;
        
    4: // Завершение
        L_Timer(IN := TRUE);
        IF L_Timer.Q THEN
            L_Timer(IN := FALSE);
            VO_Done := TRUE;
            L_State := 0;
        END_IF;
END_CASE;

END_FUNCTION_BLOCK

// POUs/FB_State_Manager
FUNCTION_BLOCK FB_State_Manager
VAR_INPUT
    VI_System_Time_MS : UDINT;
    VI_Command : BYTE; // 1-Save, 2-Restore
    VI_Heating_Config : ST_Heating_Config;
END_VAR
VAR_OUTPUT
    VO_Heating_Config : ST_Heating_Config;
    VO_Done : BOOL;
END_VAR
VAR
    L_Saved_Heating : ST_Heating_Config;
    L_Restore_Start_Time : UDINT;
    L_Restoring : BOOL;
END_VAR

CASE VI_Command OF
    1: // Save
        L_Saved_Heating := VI_Heating_Config;
        VO_Done := TRUE;
    
    2: // Restore (Плавное восстановление за 60с - ТЗ 3.6)
        IF NOT L_Restoring THEN
            L_Restoring := TRUE;
            L_Restore_Start_Time := VI_System_Time_MS;
        END_IF;
        
        IF (VI_System_Time_MS - L_Restore_Start_Time) >= 60000 THEN
            VO_Heating_Config := L_Saved_Heating;
            L_Restoring := FALSE;
            VO_Done := TRUE;
        ELSE
            // Здесь можно реализовать интерполяцию, но для простоты восстановим в конце
            VO_Done := FALSE;
        END_IF;
END_CASE;

END_FUNCTION_BLOCK

// POUs/FB_State_Snapshot_Manager
FUNCTION_BLOCK FB_State_Snapshot_Manager
VAR_INPUT
    VI_System_Time : UDINT;
    VI_Save_Req    : BOOL;
    VI_Snapshot    : ST_State_Snapshot;
END_VAR
VAR_OUTPUT
    VO_Last_ID     : UDINT;
END_VAR
VAR
    L_Buffer : ARRAY[0..9] OF ST_State_Snapshot;
    L_Idx    : INT := 0;
END_VAR

IF VI_Save_Req THEN
    L_Buffer[L_Idx] := VI_Snapshot;
    L_Buffer[L_Idx].timestamp_ms := VI_System_Time;
    VO_Last_ID := VI_System_Time;
    L_Idx := (L_Idx + 1) MOD 10;
END_IF;

END_FUNCTION_BLOCK

// POUs/FB_State_Snapshot_NVRAM
FUNCTION_BLOCK FB_State_Snapshot_NVRAM
VAR_INPUT
    VI_Command          : BYTE; // 1=SAVE, 2=LOAD
    VI_Snapshot_Ptr     : POINTER TO ST_State_Snapshot;
    VI_System_Time_MS   : UDINT;
    VI_Operator_ID      : STRING(10);
    VI_IsActivePLC      : BOOL;
    VI_TwoPersonConfirmation : BOOL;
END_VAR
VAR_OUTPUT
    VO_Done             : BOOL;
    VO_Error            : UDINT;
    VO_HMI_Status_Message : STRING(200);
END_VAR
VAR
    L_state             : BYTE;
    L_step              : UDINT;
    L_temp_buffer       : ARRAY[1..132] OF BYTE;
    L_byte_ptr          : POINTER TO BYTE;
    L_i                 : UDINT;
END_VAR
VAR CONSTANT
    C_RECORD_SIZE       : UDINT := 128;
END_VAR

// Исправленное копирование структуры через указатель
IF VI_Snapshot_Ptr <> 0 THEN
    L_byte_ptr := ADR(VI_Snapshot_Ptr^);
    
    CASE L_state OF
        1: // СОХРАНЕНИЕ (SAVE)
            IF L_step = 0 THEN
                // Копируем всю структуру байт за байтом в буфер NVRAM
                // Используем SIZEOF(ST_State_Snapshot), чтобы не выйти за границы структуры
                FOR L_i := 0 TO (SIZEOF(ST_State_Snapshot) - 1) DO
                    IF L_i < C_RECORD_SIZE THEN
                        L_temp_buffer[L_i + 1] := L_byte_ptr[TO_INT(L_i)];
                    END_IF;
                END_FOR;
                L_step := 1;
            END_IF;
            
        2: // ЗАГРУЗКА (LOAD)
            IF L_step = 2 THEN
                // Копируем из буфера обратно в структуру
                FOR L_i := 0 TO (SIZEOF(ST_State_Snapshot) - 1) DO
                    IF L_i < C_RECORD_SIZE THEN
                        L_byte_ptr[TO_INT(L_i)] := L_temp_buffer[L_i + 1];
                    END_IF;
                END_FOR;
                VO_Done := TRUE;
                L_state := 0;
            END_IF;
    END_CASE;
END_IF;

END_FUNCTION_BLOCK

// POUs/FB_Supply_Ventilation_Controller
FUNCTION_BLOCK FB_Supply_Ventilation_Controller
VAR_INPUT
    VI_Fire_Alarm : BOOL;
    VI_Gas_Alarm  : BOOL;
END_VAR
VAR_OUTPUT
    VO_Fan_Speed : BYTE;
END_VAR

IF VI_Fire_Alarm THEN
    VO_Fan_Speed := 0; // Остановка при пожаре
ELSIF VI_Gas_Alarm THEN
    VO_Fan_Speed := 100; // Максимум при утечке газа
ELSE
    VO_Fan_Speed := 40;
END_IF;

END_FUNCTION_BLOCK

// POUs/FB_Trend_Analyzer
FUNCTION_BLOCK FB_Trend_Analyzer
VAR_INPUT
    VI_Value : REAL;
    VI_Threshold_Percent : REAL := 10.0;
    VI_System_Time_MS : UDINT;
END_VAR
VAR_OUTPUT
    VO_Anomaly_Detected : BOOL;
    VO_Average_7D : REAL; // ТЗ 12.1: Скользящее среднее 7 дней
    VO_Diag_Label : BOOL; // ТЗ 12.1: Метка "диагностика"
END_VAR
VAR
    L_History : ARRAY[1..168] OF REAL; // Почасовые замеры на 7 дней
    L_Last_Hour_Time : UDINT;
    L_Idx : INT := 1;
    L_Sum : REAL;
    L_Count : INT;
    L_i : INT;
END_VAR

// 1. Накопление почасовой истории (ТЗ 12.1)
IF (VI_System_Time_MS - L_Last_Hour_Time) >= 3600000 OR L_Last_Hour_Time = 0 THEN
    L_Last_Hour_Time := VI_System_Time_MS;
    L_History[L_Idx] := VI_Value;
    L_Idx := (L_Idx MOD 168) + 1;
    IF L_Count < 168 THEN L_Count := L_Count + 1; END_IF;
END_IF;

// 2. Расчет среднего за 7 дней
L_Sum := 0.0;
IF L_Count > 0 THEN
    FOR L_i := 1 TO L_Count DO L_Sum := L_Sum + L_History[L_i]; END_FOR;
    VO_Average_7D := L_Sum / TO_REAL(L_Count);
END_IF;

// 3. Детекция аномалий и метка диагностики (ТЗ 12.1)
IF VO_Average_7D > 0.0 THEN
    VO_Anomaly_Detected := (ABS(VI_Value - VO_Average_7D) / VO_Average_7D * 100.0) > VI_Threshold_Percent;
    VO_Diag_Label := VO_Anomaly_Detected; // Метка ставится при отклонении
END_IF;

END_FUNCTION_BLOCK

// POUs/FB_TwoFactor_Auth
FUNCTION_BLOCK FB_TwoFactor_Auth
VAR_INPUT
    VI_System_Time_MS : UDINT;
    VI_Start_Auth     : BOOL;
    VI_RFID_Tag       : STRING(20);
    VI_TOTP_Code      : STRING(6);
END_VAR
VAR_OUTPUT
    VO_Auth_Passed    : BOOL;
    VO_Auth_Failed    : BOOL;
    VO_Busy           : BOOL;
END_VAR
VAR
    L_State : BYTE; // 0=Idle, 1=WaitRFID, 2=WaitTOTP
    L_Start_Timestamp : UDINT;
END_VAR

CASE L_State OF
    0: 
        IF VI_Start_Auth THEN
            L_State := 1;
            L_Start_Timestamp := VI_System_Time_MS;
            VO_Busy := TRUE;
        END_IF;
    1:
        IF VI_RFID_Tag <> '' THEN
            L_State := 2;
        ELSIF (VI_System_Time_MS - L_Start_Timestamp) > 30000 THEN
            L_State := 0;
            VO_Auth_Failed := TRUE;
            VO_Busy := FALSE;
        END_IF;
    2:
        IF VI_TOTP_Code <> '' THEN
            VO_Auth_Passed := TRUE;
            L_State := 0;
            VO_Busy := FALSE;
        END_IF;
END_CASE;

END_FUNCTION_BLOCK

// POUs/FB_Valve_Test
FUNCTION_BLOCK FB_Valve_Test
VAR_INPUT
    VI_System_Time : UDINT;
    VI_Start_Test  : BOOL;
    VI_Current_A   : REAL;
    VI_Config      : ST_Valve_Test_Config; // ТЗ 12.2
END_VAR
VAR_OUTPUT
    VO_Test_Active : BOOL;
    VO_Test_Passed : BOOL;
    VO_Deviation_Percent : REAL; // ТЗ 12.2
    VO_Error_Code : WORD;
END_VAR
VAR
    L_Start_Timestamp : UDINT;
    L_Peak_Current : REAL;
    L_Reaction_Time : UDINT;
END_VAR

IF VI_Start_Test AND NOT VO_Test_Active THEN
    VO_Test_Active := TRUE;
    L_Start_Timestamp := VI_System_Time;
    L_Peak_Current := 0.0;
    L_Reaction_Time := 0;
END_IF;

IF VO_Test_Active THEN
    IF VI_Current_A > L_Peak_Current THEN L_Peak_Current := VI_Current_A; END_IF;
    
    // Определение времени реакции (ток превысил 100мА)
    IF L_Reaction_Time = 0 AND VI_Current_A > 100.0 THEN
        L_Reaction_Time := VI_System_Time - L_Start_Timestamp;
    END_IF;

    IF (VI_System_Time - L_Start_Timestamp) > 15000 THEN
        VO_Test_Active := FALSE;
        
        // ТЗ 12.2: Контроль отклонения > 30% от номинала
        VO_Deviation_Percent := ABS(L_Peak_Current - VI_Config.Nominal_Current) / VI_Config.Nominal_Current * 100.0;
        
        VO_Test_Passed := (VO_Deviation_Percent <= 30.0) AND (L_Reaction_Time < 5000);
        
        IF NOT VO_Test_Passed THEN
            VO_Error_Code := 16#E122; // Valve Test Failed
        END_IF;
    END_IF;
END_IF;

END_FUNCTION_BLOCK

// POUs/FB_Water_Valve_Controller
FUNCTION_BLOCK FB_Water_Valve_Controller IMPLEMENTS IValveController
VAR_INPUT
    VI_IsActivePLC : BOOL;
    VI_Valve_Type : E_VALVE_TYPE;
    VI_Current_Feedback : REAL; // Ток двигателя
    VI_Limit_Open : BOOL; // Концевик открыто
    VI_Limit_Closed : BOOL; // Концевик закрыто
    VI_System_Time : UDINT;
END_VAR
VAR_OUTPUT
    VO_Valve_Open_Cmd : BOOL;
    VO_Valve_Close_Cmd : BOOL;
    VO_Status : BYTE; // 0-Open, 1-Closed, 2-Moving, 3-Error
END_VAR
VAR
    L_Moving : BOOL;
    L_Move_Start_Time : UDINT;
    L_Target_State : BOOL; // FALSE-Open, TRUE-Close
END_VAR

// Логика диагностики (п. 4.3 ТЗ)
IF L_Moving THEN
    IF (VI_System_Time - L_Move_Start_Time) > 10000 THEN // Таймаут 10 сек
        VO_Status := 3; // Ошибка
        L_Moving := FALSE;
    ELSIF (L_Target_State = TRUE AND VI_Limit_Closed) OR (L_Target_State = FALSE AND VI_Limit_Open) THEN
        VO_Status := SEL(L_Target_State, 0, 1);
        L_Moving := FALSE;
    ELSE
        VO_Status := 2; // Moving
    END_IF;
END_IF;

METHOD CloseValve : BOOL
VAR_INPUT
    VI_Operator_ID : STRING(10);
    VI_Force : BOOL;
END_VAR
IF VI_IsActivePLC OR VI_Force THEN
    VO_Valve_Open_Cmd := FALSE;
    VO_Valve_Close_Cmd := TRUE;
    L_Moving := TRUE;
    L_Target_State := TRUE;
    L_Move_Start_Time := VI_System_Time;
    CloseValve := TRUE;
ELSE
    CloseValve := FALSE;
END_IF;
END_METHOD

METHOD GetStatus : BYTE
VAR_INPUT
END_VAR
GetStatus := VO_Status;
END_METHOD

METHOD OpenValve : BOOL
VAR_INPUT
    VI_Operator_ID : STRING(10);
    VI_Force : BOOL;
END_VAR
IF VI_IsActivePLC OR VI_Force THEN
    VO_Valve_Open_Cmd := TRUE;
    VO_Valve_Close_Cmd := FALSE;
    L_Moving := TRUE;
    L_Target_State := FALSE;
    L_Move_Start_Time := VI_System_Time;
    OpenValve := TRUE;
ELSE
    OpenValve := FALSE;
END_IF;
END_METHOD

END_FUNCTION_BLOCK

// POUs/FB_Zone_Access_Manager
FUNCTION_BLOCK FB_Zone_Access_Manager
VAR_INPUT
    VI_Operator_ID : STRING(10);
    VI_Zone_ID     : BYTE;
    VI_Req_Level   : BYTE;
END_VAR
VAR
    L_Rights : ARRAY[1..10] OF ST_Operator_Zone_Rights;
END_VAR

METHOD CheckAccess : BOOL
VAR_INPUT
    VI_Op : STRING(10);
    VI_Req_Level : BYTE;
END_VAR
IF VI_Op = 'ADMIN' THEN
    // Если 2FA включена, проверяем флаг прохождения второго фактора
    IF GVL_HMI_Config.G_HMI_Admin_2FA_Enabled THEN
        CheckAccess := GVL_HMI_Config.G_HMI_Current_Operator_Factor2_Done;
    ELSE
        CheckAccess := TRUE;
    END_IF;
ELSIF VI_Op = 'SERVICE' AND VI_Req_Level <= 3 THEN
    CheckAccess := TRUE;
ELSE
    CheckAccess := FALSE;
END_IF;
END_METHOD

END_FUNCTION_BLOCK

// /Visualization
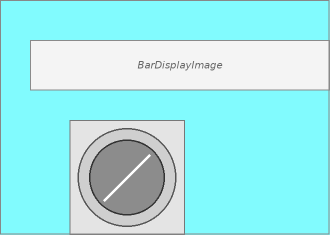
VISUALIZATION Visualization  // 330x235, background image 
    BarDisplayImage (30,40 300x50), value: AI_DHW_Temp, style: BarDisplayImage-gray, scale format: %.1f, scale 0..100
    Potentiometer360 (40,120 174x115), variable: AI_DHW_Temp, style: Potentiometer-Potentiometer360-Gray, scale format: %.1f, scale 0..100
        p2431819421: Outside
END_VISUALIZATION
